// TIA Portal V19 export
TYPE "MatCountCOut"
// stored: Access Published
   STRUCT
      AlarmsPresence : Bool;
      WarningPresence : Bool;
      CounterValid : Bool;
      Standstill : Bool;
      PresetDone : Bool;
      CounterValue : LReal;
      EncoderPosValue : LReal;
      FAK : LReal;
      AX_MODULE : LReal;
      COUNTER_MODULE : LReal;
   END_STRUCT;
END_TYPE
